INTERFACE I_Interface2

END_INTERFACE

(* stored: Version 1.1.0.1, ProductVersion 3.1.4024.3
   Itf I_Interface2: Id {386f884a-1f12-4cc9-b963-c0257e353c99} *)
